{attribute 'qualified_only'}
VAR_GLOBAL
	
	// outputs
	TurnTableMotorTurn AT %Q* : BOOL;
	TurnTableMotorReverse AT %Q* : BOOL;
	ConvaorbeltMotorRun AT %Q* : BOOL;
	ConvaorbeltMotorReverse AT %Q* : BOOL;
	QuittierenLamp AT %Q* : BOOL;
	OnOffStatusLamp AT %Q* : BOOL;

	// inputs
	StartButton AT %I* : BOOL;
	StopButton AT %I* : BOOL;
	EmStop AT %I* : BOOL;
	ResetButton AT %I* : BOOL;
	
	
END_VAR

(* stored: Version 1.1.0.1
   GVL InputOutput: Id {3bfff44a-42d8-4e67-8a72-cea7f144b7e9} *)
